FUNCTION_BLOCK FB_Restore
VAR_INPUT
	bEnable : BOOL;
	iMotorPrev 		: 	INT;
	eStep		:	E_Step;
	eSubStepSensor	:	E_Step;
	eSubStepPistons	:	E_Step;
END_VAR
VAR_IN_OUT
	stIn		:	ST_CSL_In;
	stParams	: 	ST_CSL_Params;
	stOut		:	ST_CSL_Out;
END_VAR
VAR_OUTPUT
	bFbEnd		:	BOOL;
END_VAR
VAR
	iMotor		:	INT;

	bPieceOut 	:	BOOL;	

	fbRtMotorImpulse : R_TRIG;
	
	bInitialized: BOOL;
END_VAR


IF NOT bInitialized THEN
	bFbEnd := FALSE;
	bInitialized := TRUE;
	bPieceOut := FALSE;
	iMotor := 0;
ELSE
	IF eSubStepSensor = e_Step.Start THEN
		bInitialized := FALSE;
		bFbEnd := TRUE;
	END_IF
	IF eStep = E_Step.MainSensor AND NOT bPieceOut THEN
		stOut.bMotor := TRUE;
		IF NOT stIn.bPieceSensorOutput AND bEnable THEN
			bPieceOut := TRUE;
			iMotor := 0;
		END_IF	
	ELSIF eStep = E_Step.MainPiston  OR bPieceOut THEN
		stOut.bMotor := TRUE;
	
		fbRtMotorImpulse(CLK:=	stIn.bMotorImpulse );
		
		IF fbRtMotorImpulse.Q	THEN
			iMotor := iMotor + 1;
		END_IF
			
		IF (iMotor >= (stParams.StepNoSlot - iMotorPrev)  AND eStep = E_Step.MainPiston) OR (iMotor = stParams.StepNoSlot AND eStep = E_Step.MainSensor) THEN
			stOut.bMotor := FALSE;
			bInitialized := FALSE;
			bFbEnd := TRUE;		
		END_IF

	ELSE
		bInitialized := FALSE;
		bFbEnd := TRUE;
	END_IF
END_IF

END_FUNCTION_BLOCK

(* stored: Version 1.1.0.1, ProductVersion 3.1.4024.12
   POU FB_Restore: Id {fd15dcd7-03bd-4602-ba28-f37f0729ceb4}, SpecialFunc None *)
